// Dublê de teste de FB_DfiDbWriter: sobrescreve apenas o seam DoExecute,
// deixando toda a maquina de estados da classe base rodar de verdade.
// FB_SQLCommandEvt/FB_SQLDatabaseEvt exigem um TwinCAT Database Server real,
// por isso o caminho de banco nao e coberto aqui (bancada, Task 15).
FUNCTION_BLOCK FB_DfiDbWriter_Fake EXTENDS FB_DfiDbWriter
VAR
	nScript    : INT;
	nExecCycle : INT;
END_VAR
VAR CONSTANT
	// Espelhadas em FB_DfiDbWriter_Tests (VAR CONSTANT de FB nao e visivel de
	// fora da instancia). Manter os dois blocos em sincronia.
	SCRIPT_OK         : INT := 1;
	SCRIPT_EXEC_ERROR : INT := 2;
	SCRIPT_DB_LOST    : INT := 3;
END_VAR

// A maquina de estados da base vive no metodo herdado Cycle() (nao
// sobrescrito). Chamado aqui em vez de SUPER^() porque VAR_IN_OUT (fbBuffer)
// nao pode ser religado num SUPER^(). DoExecute/DoConnect continuam
// despachando para os overrides deste fake.
Cycle();

METHOD SetScript
VAR_INPUT
	n : INT;
END_VAR
nScript    := n;
nExecCycle := 0;
// Pula o estado CONNECT: os testes exercitam BUILD/EXECUTE/COMMIT direto.
bDbConnected := TRUE;
eState       := E_DfiWriterState.IDLE;
END_METHOD

METHOD PROTECTED DoConnect : INT
// O fake nunca fala com um banco real: conecta instantaneamente.
// 0 = ocupado, 1 = conectado e comando criado, 2 = erro (mesmo contrato da base).
DoConnect := 1;
END_METHOD

METHOD PROTECTED DoExecute : INT
// 0 = ocupado, 1 = ok, 2 = erro (mesmo contrato do metodo sobrescrito).
IF nScript = SCRIPT_EXEC_ERROR THEN
	DoExecute := 2;

ELSIF nScript = SCRIPT_DB_LOST THEN
	// conexao cai no meio do Execute: a base deve ir para DB_LOST sem Pop
	bDbConnected := FALSE;
	DoExecute := 0;

ELSIF nScript = SCRIPT_OK THEN
	// 1 ciclo "ocupado" e depois sucesso, para exercitar a espera em EXECUTE
	IF nExecCycle = 0 THEN
		nExecCycle := 1;
		DoExecute := 0;
	ELSE
		DoExecute := 1;
	END_IF

ELSE
	DoExecute := 1;
END_IF
END_METHOD

END_FUNCTION_BLOCK

(* stored: Version 1.1.0.1
   POU FB_DfiDbWriter_Fake: Id {2d93a3b7-760e-4042-9461-eb2d104b1435}, SpecialFunc None
   Method SetScript: Id {5a7dc5b0-bb30-47f9-b8e6-a3eff9d86101}
   Method DoConnect: Id {fbbf006d-c49b-40ee-82e7-abe446e62729}
   Method DoExecute: Id {53ec1518-e2e5-4d33-ac7e-26f6dce9806b} *)
